(* Logix 5000 project; controller remote_controller Emulate 5570 rev 30.12; software revision 30.01 *)

TASK MainTask (continuous, watchdog 500 ms) : MainProgram

MODULES
   Local : Emulate 5570 (ICP 4, rev 30.12)
      PLC01_Traffic_Light_Limits : Emulate 5570 (ICP 2, rev 30.1)   // conexion between two plc
END_MODULES

VAR_GLOBAL   (* controller tags *)
   Messages_Data : DINT;
   RRemote : DINT; {produced}
        .0   // critical process sensor
END_VAR

PROGRAM MainProgram   (* main routine MainRoutine *)

ROUTINE MainRoutine   (* ladder *)
END_ROUTINE
END_PROGRAM
